Staubli VAL3: decodeDesc.pgx

program decodeDesc(mdesc& value, num& buffer[])
  local num decodeBuffer[3]
begin
  fromBinary(buffer, 8, "4.0b", decodeBuffer)

  value.tvel = decodeBuffer[0]
  value.rvel = decodeBuffer[1]

  fromBinary(buffer[8], 3, "1", decodeBuffer)
  value.accel = decodeBuffer[0]
  value.vel   = decodeBuffer[1]
  value.decel = decodeBuffer[2]

  logMsg("D: (" + toString("3", value.tvel) + ", " + toString("3", value.rvel) + ", " + toString("3", value.accel) + ", " + toString("3", value.vel) + ", " + toString("3", value.decel) + ")")
end
